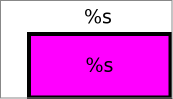
VISUALIZATION Obj_Energy_Meter  // 173x99
VAR_INPUT
	sIndex : STRING;
	bStatus : WORD;
	bOffline : BOOL;
	fOperating_Hrs : REAL;
	fEnergy : REAL;
	fVolume : REAL;
	fSupply_Temp : REAL;
	fReturn_Temp : REAL;
	fTemp_Diff :REAL;
END_VAR
    Rectangle (27,32 145x67), "%s", colour toggle: (bStatus =1) OR (bStatus = 2), text list: 'Energy_Meters_Status', text index: bStatus
        OnMouseClick: OpenDialog Dialog=Dialog_EnergyMeter, Parameters={fEnergy: fEnergy, fOperHours: fOperating_Hrs, fReturn_Temp: fReturn_Temp, fSupply_Temp: fSupply_Temp, fTemp_Diff: fTemp_Diff, fVolume: fVolume, sHeader: sIndex}, OpenModal=True, OpenCentered=True
    Rectangle (23,2 150x30), "%s", text variable: sIndex
    Rectangle (27,32 145x67), "%s", invisible if: Not bOffline, text list: 'Energy_Meters_Status', text index: bStatus
END_VISUALIZATION

(* stored: Version 1.1.0.1, ProductVersion 3.1.4024.12
   Visu Obj_Energy_Meter: Id {cd2a10d7-a64f-4c80-8416-5dbc6c390954} *)
